					END_IF
				END_IF
			END_IF
			IF GVL.mb_Output_Coils[GVL.REALTIME_RETARD] THEN
				IF GVL_IO.LateralMotorPot[FTN6] > 800 THEN				//test the FB for limit - assumes 32767 is max of 10 VDC
					GVL_IO.LateralMotorRelay[FTN6,GVL.iPlus] := FALSE;				// turn on the reverse output
					GVL_IO.LateralMotorRelay[FTN6,GVL.iMinus] := TRUE;
					wCycleCount := wCycleCount + 1;
					IF (wCycleCount > wMotorTimeOn) OR GVL_IO.LateralMotorLimit[FTN6,GVL.iPlus] OR
							GVL_IO.LateralMotorLimit[FTN6,GVL.iMinus] THEN	//done with timer or any limit activated
						GVL_IO.LateralMotorRelay[FTN6,GVL.iPlus] := FALSE;		//turn off outputs
						GVL_IO.LateralMotorRelay[FTN6,GVL.iMinus] := FALSE;
						GVL.mb_Output_Coils[GVL.REALTIME_RETARD] := FALSE; // reset the reverse boolean
						wCycleCount := 0;					//reset the timer counter						
						nRawFBpos	:=	GVL_IO.LateralMotorPot[FTN6];
						nActualPos		:= 	LREAL_TO_DINT(
							INT_TO_LREAL(GVL.w_RegisterConfig[Index,GVL.iLAT,0 ]) +							//base is min position
							(((INT_TO_LREAL(nRawFBpos - GVL.w_RegisterConfig[Index,GVL.iLAT,2 ])) 			//voltage offset from low calibration
							* 	(INT_TO_LREAL(GVL.w_RegisterConfig[Index,GVL.iLAT,1 ] - GVL.w_RegisterConfig[Index,GVL.iLAT,0 ])))	//total position length
							/	( INT_TO_LREAL(GVL.w_RegisterConfig[Index,GVL.iLAT,3 ] - GVL.w_RegisterConfig[Index,GVL.iLAT,2 ])))	//total voltage range
							);
						GVL.mb_Output_Registers[w_temp_index+(GVL.iActualPosition)]	:= 
								DINT_TO_WORD(nActualPos);		//post the scaled actual position here to OUTPUT
					END_IF
				END_IF
			END_IF
	 38:	//Lateral FB Ftn 7
			GVL.mb_Output_Registers[GVL.REALTIME_PLC_A2D] :=	INT_TO_WORD(GVL_IO.LateralMotorPot[FTN7]);
			w_temp_index	:= GVL.RUNREG_START+(GVL.RUNREG_SIZE*3*FTN7)+(GVL.RUNREG_SIZE*GVL.iLAT)+10;
			IF GVL.mb_Output_Coils[GVL.REALTIME_ADVANCE] THEN		//move the motor forward
				IF GVL_IO.LateralMotorPot[FTN7] < 32000 THEN				//test the FB for limit - assumes 32767 is max of 10 VDC
					GVL_IO.LateralMotorRelay[FTN7,GVL.iPlus] := TRUE;				// turn on the advance output
					GVL_IO.LateralMotorRelay[FTN7,GVL.iMinus] := FALSE;
					wCycleCount := wCycleCount + 1;
					IF (wCycleCount > wMotorTimeOn) OR GVL_IO.LateralMotorLimit[FTN7,GVL.iPlus] OR
							GVL_IO.LateralMotorLimit[FTN7,GVL.iMinus] THEN	//done with timer or any limit activated
						GVL_IO.LateralMotorRelay[FTN7,GVL.iPlus] := FALSE;		//turn off outputs
						GVL_IO.LateralMotorRelay[FTN7,GVL.iMinus] := FALSE;
						GVL.mb_Output_Coils[GVL.REALTIME_ADVANCE] := FALSE; // reset the advance boolean
						wCycleCount := 0;					//reset the timer counter						
						nRawFBpos	:=	GVL_IO.LateralMotorPot[FTN7];
						nActualPos		:= 	LREAL_TO_DINT(
							INT_TO_LREAL(GVL.w_RegisterConfig[Index,GVL.iLAT,0 ]) +							//base is min position
							(((INT_TO_LREAL(nRawFBpos - GVL.w_RegisterConfig[Index,GVL.iLAT,2 ])) 			//voltage offset from low calibration
							* 	(INT_TO_LREAL(GVL.w_RegisterConfig[Index,GVL.iLAT,1 ] - GVL.w_RegisterConfig[Index,GVL.iLAT,0 ])))	//total position length
							/	( INT_TO_LREAL(GVL.w_RegisterConfig[Index,GVL.iLAT,3 ] - GVL.w_RegisterConfig[Index,GVL.iLAT,2 ])))	//total voltage range
							);
						GVL.mb_Output_Registers[w_temp_index+(GVL.iActualPosition)]	:= 
								DINT_TO_WORD(nActualPos);		//post the scaled actual position here to OUTPUT

					END_IF
				END_IF
			END_IF
			IF GVL.mb_Output_Coils[GVL.REALTIME_RETARD] THEN
				IF GVL_IO.LateralMotorPot[FTN7] > 800 THEN				//test the FB for limit - assumes 32767 is max of 10 VDC
					GVL_IO.LateralMotorRelay[FTN7,GVL.iPlus] := FALSE;				// turn on the reverse output
					GVL_IO.LateralMotorRelay[FTN7,GVL.iMinus] := TRUE;
					wCycleCount := wCycleCount + 1;
					IF (wCycleCount > wMotorTimeOn) OR GVL_IO.LateralMotorLimit[FTN7,GVL.iPlus] OR
							GVL_IO.LateralMotorLimit[FTN7,GVL.iMinus] THEN	//done with timer or any limit activated
						GVL_IO.LateralMotorRelay[FTN7,GVL.iPlus] := FALSE;		//turn off outputs
						GVL_IO.LateralMotorRelay[FTN7,GVL.iMinus] := FALSE;
						GVL.mb_Output_Coils[GVL.REALTIME_RETARD] := FALSE; // reset the reverse boolean
						wCycleCount := 0;					//reset the timer counter						
						nRawFBpos	:=	GVL_IO.LateralMotorPot[FTN7];
						nActualPos		:= 	LREAL_TO_DINT(
							INT_TO_LREAL(GVL.w_RegisterConfig[Index,GVL.iLAT,0 ]) +							//base is min position
							(((INT_TO_LREAL(nRawFBpos - GVL.w_RegisterConfig[Index,GVL.iLAT,2 ])) 			//voltage offset from low calibration
							* 	(INT_TO_LREAL(GVL.w_RegisterConfig[Index,GVL.iLAT,1 ] - GVL.w_RegisterConfig[Index,GVL.iLAT,0 ])))	//total position length
							/	( INT_TO_LREAL(GVL.w_RegisterConfig[Index,GVL.iLAT,3 ] - GVL.w_RegisterConfig[Index,GVL.iLAT,2 ])))	//total voltage range
							);
						GVL.mb_Output_Registers[w_temp_index+(GVL.iActualPosition)]	:= 
								DINT_TO_WORD(nActualPos);		//post the scaled actual position here to OUTPUT
					END_IF
				END_IF
			END_IF
	 39:	//Lateral FB Ftn 8
			GVL.mb_Output_Registers[GVL.REALTIME_PLC_A2D] :=	INT_TO_WORD(GVL_IO.LateralMotorPot[FTN8]);
			w_temp_index	:= GVL.RUNREG_START+(GVL.RUNREG_SIZE*3*FTN8)+(GVL.RUNREG_SIZE*GVL.iLAT)+10;
			IF GVL.mb_Output_Coils[GVL.REALTIME_ADVANCE] THEN		//move the motor forward
				IF GVL_IO.LateralMotorPot[FTN8] < 32000 THEN				//test the FB for limit - assumes 32767 is max of 10 VDC
					GVL_IO.LateralMotorRelay[FTN8,GVL.iPlus] := TRUE;				// turn on the advance output
					GVL_IO.LateralMotorRelay[FTN8,GVL.iMinus] := FALSE;
					wCycleCount := wCycleCount + 1;
					IF (wCycleCount > wMotorTimeOn) OR GVL_IO.LateralMotorLimit[FTN8,GVL.iPlus] OR
							GVL_IO.LateralMotorLimit[FTN8,GVL.iMinus] THEN	//done with timer or any limit activated
						GVL_IO.LateralMotorRelay[FTN8,GVL.iPlus] := FALSE;		//turn off outputs
						GVL_IO.LateralMotorRelay[FTN8,GVL.iMinus] := FALSE;
						GVL.mb_Output_Coils[GVL.REALTIME_ADVANCE] := FALSE; // reset the advance boolean
						wCycleCount := 0;					//reset the timer counter						
						nRawFBpos	:=	GVL_IO.LateralMotorPot[FTN8];
						nActualPos		:= 	LREAL_TO_DINT(
							INT_TO_LREAL(GVL.w_RegisterConfig[Index,GVL.iLAT,0 ]) +							//base is min position
							(((INT_TO_LREAL(nRawFBpos - GVL.w_RegisterConfig[Index,GVL.iLAT,2 ])) 			//voltage offset from low calibration
							* 	(INT_TO_LREAL(GVL.w_RegisterConfig[Index,GVL.iLAT,1 ] - GVL.w_RegisterConfig[Index,GVL.iLAT,0 ])))	//total position length
							/	( INT_TO_LREAL(GVL.w_RegisterConfig[Index,GVL.iLAT,3 ] - GVL.w_RegisterConfig[Index,GVL.iLAT,2 ])))	//total voltage range
							);
						GVL.mb_Output_Registers[w_temp_index+(GVL.iActualPosition)]	:= 
								DINT_TO_WORD(nActualPos);		//post the scaled actual position here to OUTPUT

					END_IF
				END_IF
			END_IF
			IF GVL.mb_Output_Coils[GVL.REALTIME_RETARD] THEN
				IF GVL_IO.LateralMotorPot[FTN8] > 800 THEN				//test the FB for limit - assumes 32767 is max of 10 VDC
					GVL_IO.LateralMotorRelay[FTN8,GVL.iPlus] := FALSE;				// turn on the reverse output
					GVL_IO.LateralMotorRelay[FTN8,GVL.iMinus] := TRUE;
					wCycleCount := wCycleCount + 1;
					IF (wCycleCount > wMotorTimeOn) OR GVL_IO.LateralMotorLimit[FTN8,GVL.iPlus] OR
							GVL_IO.LateralMotorLimit[FTN8,GVL.iMinus] THEN	//done with timer or any limit activated
						GVL_IO.LateralMotorRelay[FTN8,GVL.iPlus] := FALSE;		//turn off outputs
						GVL_IO.LateralMotorRelay[FTN8,GVL.iMinus] := FALSE;
						GVL.mb_Output_Coils[GVL.REALTIME_RETARD] := FALSE; // reset the reverse boolean
						wCycleCount := 0;					//reset the timer counter						
						nRawFBpos	:=	GVL_IO.LateralMotorPot[FTN8];
						nActualPos		:= 	LREAL_TO_DINT(
							INT_TO_LREAL(GVL.w_RegisterConfig[Index,GVL.iLAT,0 ]) +							//base is min position
							(((INT_TO_LREAL(nRawFBpos - GVL.w_RegisterConfig[Index,GVL.iLAT,2 ])) 			//voltage offset from low calibration
							* 	(INT_TO_LREAL(GVL.w_RegisterConfig[Index,GVL.iLAT,1 ] - GVL.w_RegisterConfig[Index,GVL.iLAT,0 ])))	//total position length
							/	( INT_TO_LREAL(GVL.w_RegisterConfig[Index,GVL.iLAT,3 ] - GVL.w_RegisterConfig[Index,GVL.iLAT,2 ])))	//total voltage range
							);
						GVL.mb_Output_Registers[w_temp_index+(GVL.iActualPosition)]	:= 
								DINT_TO_WORD(nActualPos);		//post the scaled actual position here to OUTPUT
					END_IF
				END_IF
			END_IF
	 40:	//Lateral FB Ftn 9
			GVL.mb_Output_Registers[GVL.REALTIME_PLC_A2D] :=	INT_TO_WORD(GVL_IO.LateralMotorPot[FTN9]);
			w_temp_index	:= GVL.RUNREG_START+(GVL.RUNREG_SIZE*3*FTN9)+(GVL.RUNREG_SIZE*GVL.iLAT)+10;
			IF GVL.mb_Output_Coils[GVL.REALTIME_ADVANCE] THEN		//move the motor forward
				IF GVL_IO.LateralMotorPot[FTN9] < 32000 THEN				//test the FB for limit - assumes 32767 is max of 10 VDC
					GVL_IO.LateralMotorRelay[FTN9,GVL.iPlus] := TRUE;				// turn on the advance output
					GVL_IO.LateralMotorRelay[FTN9,GVL.iMinus] := FALSE;
					wCycleCount := wCycleCount + 1;
					IF (wCycleCount > wMotorTimeOn) OR GVL_IO.LateralMotorLimit[FTN9,GVL.iPlus] OR
							GVL_IO.LateralMotorLimit[FTN9,GVL.iMinus] THEN	//done with timer or any limit activated
						GVL_IO.LateralMotorRelay[FTN9,GVL.iPlus] := FALSE;		//turn off outputs
						GVL_IO.LateralMotorRelay[FTN9,GVL.iMinus] := FALSE;
						GVL.mb_Output_Coils[GVL.REALTIME_ADVANCE] := FALSE; // reset the advance boolean
						wCycleCount := 0;					//reset the timer counter						
						nRawFBpos	:=	GVL_IO.LateralMotorPot[FTN9];
						nActualPos		:= 	LREAL_TO_DINT(
							INT_TO_LREAL(GVL.w_RegisterConfig[Index,GVL.iLAT,0 ]) +							//base is min position
							(((INT_TO_LREAL(nRawFBpos - GVL.w_RegisterConfig[Index,GVL.iLAT,2 ])) 			//voltage offset from low calibration
							* 	(INT_TO_LREAL(GVL.w_RegisterConfig[Index,GVL.iLAT,1 ] - GVL.w_RegisterConfig[Index,GVL.iLAT,0 ])))	//total position length
							/	( INT_TO_LREAL(GVL.w_RegisterConfig[Index,GVL.iLAT,3 ] - GVL.w_RegisterConfig[Index,GVL.iLAT,2 ])))	//total voltage range
							);
						GVL.mb_Output_Registers[w_temp_index+(GVL.iActualPosition)]	:= 
								DINT_TO_WORD(nActualPos);		//post the scaled actual position here to OUTPUT

					END_IF
				END_IF
			END_IF
			IF GVL.mb_Output_Coils[GVL.REALTIME_RETARD] THEN
				IF GVL_IO.LateralMotorPot[FTN9] > 800 THEN				//test the FB for limit - assumes 32767 is max of 10 VDC
					GVL_IO.LateralMotorRelay[FTN9,GVL.iPlus] := FALSE;				// turn on the reverse output
					GVL_IO.LateralMotorRelay[FTN9,GVL.iMinus] := TRUE;
					wCycleCount := wCycleCount + 1;
					IF (wCycleCount > wMotorTimeOn) OR GVL_IO.LateralMotorLimit[FTN9,GVL.iPlus] OR
							GVL_IO.LateralMotorLimit[FTN9,GVL.iMinus] THEN	//done with timer or any limit activated
						GVL_IO.LateralMotorRelay[FTN9,GVL.iPlus] := FALSE;		//turn off outputs
						GVL_IO.LateralMotorRelay[FTN9,GVL.iMinus] := FALSE;
						GVL.mb_Output_Coils[GVL.REALTIME_RETARD] := FALSE; // reset the reverse boolean
						wCycleCount := 0;					//reset the timer counter						
						nRawFBpos	:=	GVL_IO.LateralMotorPot[FTN9];
						nActualPos		:= 	LREAL_TO_DINT(
							INT_TO_LREAL(GVL.w_RegisterConfig[Index,GVL.iLAT,0 ]) +							//base is min position
							(((INT_TO_LREAL(nRawFBpos - GVL.w_RegisterConfig[Index,GVL.iLAT,2 ])) 			//voltage offset from low calibration
							* 	(INT_TO_LREAL(GVL.w_RegisterConfig[Index,GVL.iLAT,1 ] - GVL.w_RegisterConfig[Index,GVL.iLAT,0 ])))	//total position length
							/	( INT_TO_LREAL(GVL.w_RegisterConfig[Index,GVL.iLAT,3 ] - GVL.w_RegisterConfig[Index,GVL.iLAT,2 ])))	//total voltage range
							);
						GVL.mb_Output_Registers[w_temp_index+(GVL.iActualPosition)]	:= 
								DINT_TO_WORD(nActualPos);		//post the scaled actual position here to OUTPUT
					END_IF
				END_IF
			END_IF
	 41:	//Lateral FB Ftn 10
			GVL.mb_Output_Registers[GVL.REALTIME_PLC_A2D] :=	INT_TO_WORD(GVL_IO.LateralMotorPot[FTN10]);
			w_temp_index	:= GVL.RUNREG_START+(GVL.RUNREG_SIZE*3*FTN10)+(GVL.RUNREG_SIZE*GVL.iLAT)+10;
			IF GVL.mb_Output_Coils[GVL.REALTIME_ADVANCE] THEN		//move the motor forward
				IF GVL_IO.LateralMotorPot[FTN10] < 32000 THEN				//test the FB for limit - assumes 32767 is max of 10 VDC
					GVL_IO.LateralMotorRelay[FTN10,GVL.iPlus] := TRUE;				// turn on the advance output
					GVL_IO.LateralMotorRelay[FTN10,GVL.iMinus] := FALSE;
					wCycleCount := wCycleCount + 1;
					IF (wCycleCount > wMotorTimeOn) OR GVL_IO.LateralMotorLimit[FTN10,GVL.iPlus] OR
							GVL_IO.LateralMotorLimit[FTN10,GVL.iMinus] THEN	//done with timer or any limit activated
						GVL_IO.LateralMotorRelay[FTN10,GVL.iPlus] := FALSE;		//turn off outputs
						GVL_IO.LateralMotorRelay[FTN10,GVL.iMinus] := FALSE;
						GVL.mb_Output_Coils[GVL.REALTIME_ADVANCE] := FALSE; // reset the advance boolean
						wCycleCount := 0;					//reset the timer counter						
						nRawFBpos	:=	GVL_IO.LateralMotorPot[FTN10];
						nActualPos		:= 	LREAL_TO_DINT(
							INT_TO_LREAL(GVL.w_RegisterConfig[Index,GVL.iLAT,0 ]) +							//base is min position
							(((INT_TO_LREAL(nRawFBpos - GVL.w_RegisterConfig[Index,GVL.iLAT,2 ])) 			//voltage offset from low calibration
							* 	(INT_TO_LREAL(GVL.w_RegisterConfig[Index,GVL.iLAT,1 ] - GVL.w_RegisterConfig[Index,GVL.iLAT,0 ])))	//total position length
							/	( INT_TO_LREAL(GVL.w_RegisterConfig[Index,GVL.iLAT,3 ] - GVL.w_RegisterConfig[Index,GVL.iLAT,2 ])))	//total voltage range
							);
						GVL.mb_Output_Registers[w_temp_index+(GVL.iActualPosition)]	:= 
								DINT_TO_WORD(nActualPos);		//post the scaled actual position here to OUTPUT

					END_IF
				END_IF
			END_IF
			IF GVL.mb_Output_Coils[GVL.REALTIME_RETARD] THEN
				IF GVL_IO.LateralMotorPot[FTN10] > 800 THEN				//test the FB for limit - assumes 32767 is max of 10 VDC
					GVL_IO.LateralMotorRelay[FTN10,GVL.iPlus] := FALSE;				// turn on the reverse output
					GVL_IO.LateralMotorRelay[FTN10,GVL.iMinus] := TRUE;
					wCycleCount := wCycleCount + 1;
					IF (wCycleCount > wMotorTimeOn) OR GVL_IO.LateralMotorLimit[FTN10,GVL.iPlus] OR
							GVL_IO.LateralMotorLimit[FTN10,GVL.iMinus] THEN	//done with timer or any limit activated
						GVL_IO.LateralMotorRelay[FTN10,GVL.iPlus] := FALSE;		//turn off outputs
						GVL_IO.LateralMotorRelay[FTN10,GVL.iMinus] := FALSE;
						GVL.mb_Output_Coils[GVL.REALTIME_RETARD] := FALSE; // reset the reverse boolean
						wCycleCount := 0;					//reset the timer counter						
						nRawFBpos	:=	GVL_IO.LateralMotorPot[FTN10];
						nActualPos		:= 	LREAL_TO_DINT(
							INT_TO_LREAL(GVL.w_RegisterConfig[Index,GVL.iLAT,0 ]) +							//base is min position
							(((INT_TO_LREAL(nRawFBpos - GVL.w_RegisterConfig[Index,GVL.iLAT,2 ])) 			//voltage offset from low calibration
							* 	(INT_TO_LREAL(GVL.w_RegisterConfig[Index,GVL.iLAT,1 ] - GVL.w_RegisterConfig[Index,GVL.iLAT,0 ])))	//total position length
							/	( INT_TO_LREAL(GVL.w_RegisterConfig[Index,GVL.iLAT,3 ] - GVL.w_RegisterConfig[Index,GVL.iLAT,2 ])))	//total voltage range
							);
						GVL.mb_Output_Registers[w_temp_index+(GVL.iActualPosition)]	:= 
								DINT_TO_WORD(nActualPos);		//post the scaled actual position here to OUTPUT
					END_IF
				END_IF
			END_IF
//	 42:	//Skew FB Ftn 1 ... not yet...
	 END_CASE  // end of GVL.REALTIME_DATA_SELECTION
	 
//--------------------------------- end of Real-time support ------------------------------------------

END_FUNCTION_BLOCK

(* stored: Version 1.1.0.1, ProductVersion 3.1.4022.10
   POU FBRealtimeSupport: Id {6abeff8e-f12a-423c-ba2e-ae8ec777e99d}, SpecialFunc None *)
